(* Schneider Machine Expert - Basic project motor_starter, file version 2.2.0.0 *)
(* ProjectInformations: Name=New project *)

HARDWARE
  Cpu 0: TM221CE40R
  EthernetConfiguration: NetworkName=M221, IpAllocationMode=FixedAddress, IpAddress=0.0.0.0, SubnetMask=0.0.0.0
  SerialLineConfiguration: Baud=Baud19200, Parity=ParityEven, DataBits=DataBits8, StopBits=StopBits1, PhysicalMedium=PhysicalMediumRs485, TransmissionMode=TransmissionModeModbusRtu, SlaveId=1, Addressing=SlaveAddressing
  MastTask: UsePeriodScanMode=false, PeriodScan=100
  FastTask: Period=255
  CpuBehavior: StartingMode=StartAsPreviousState, AutoSaveRamOnEeprom=true, WatchdogPeriod=250

SYMBOLS  (address, symbol, comment, settings)
  %I0.0     I0  "Start"
  %I0.1       "Stop"
  %Q0.0     O0

POU New POU
  (* SectionNumber=1 *)

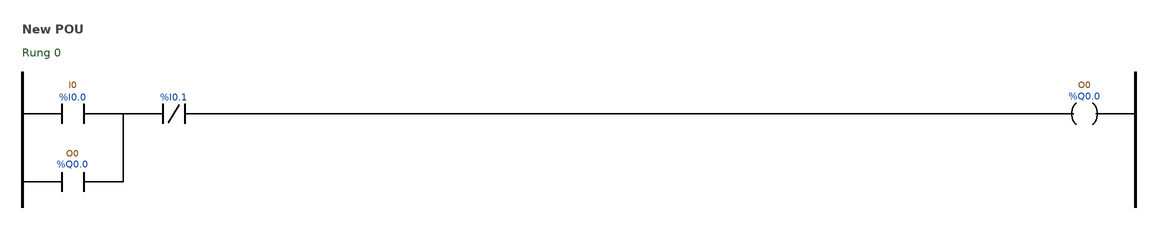

// Rung 0
  LD %I0.0                (* I0 *)
  OR %Q0.0                (* O0 *)
  ANDN %I0.1
  ST %Q0.0                (* O0 *)
  // as ST:
  //   O0 := (I0 OR O0) AND NOT %I0.1;
